// TIA Portal V17 program export: 1 tag tables, 1 data types, 1 data blocks, 3 code blocks (in call order from the OBs), 1 instance data blocks

VAR_GLOBAL   // PLC tag table "IO_CC_Cav_A"
   O_CC_Coupelle_Up_Cav_A AT %Q600.7 : Bool;
   I_CC_TyrePresent_Pos_2_Cav_A AT %I600.2 : Bool;
   I_CC_TyrePresent_Pos_3_Cav_A AT %I600.3 : Bool;
   I_CC_TyrePresent_Coupelle_Cav_A AT %I600.0 : Bool;
   I_CC_TyrePresent_Exit_Cav_A AT %I600.1 : Bool;
   I_CC_Coupelle_Low_Cav_A AT %I600.4 : Bool;
   I_CC_Coupelle_High_Cav_A AT %I600.5 : Bool;
   I_CC_Motor_Lototo_Cav_A AT %I600.6 : Bool;
   O_CC_Coupelle_Down_Cav_A AT %Q601.7 : Bool;
   I_CC_TyrePresent_Pos_1_Cav_A AT %I601.0 : Bool;
END_VAR

TYPE "CAB"
// stored: IsFailsafeCompliant false
   STRUCT
      CAB : String[20];
   END_STRUCT;
END_TYPE

DATA_BLOCK "GlobalData"   // DB1
{ S7_Optimized_Access := 'TRUE' }
VERSION : 0.1
// stored: AutoNumber true, IsIECCheckEnabled false
   VAR
      Ready : Bool;
      Count : Int;
      Config : Struct
         MaxSpeed : Real;
         Enabled : Bool;
      END_STRUCT;
   END_VAR
BEGIN
END_DATA_BLOCK

ORGANIZATION_BLOCK "Main"   // OB1, LAD, ProgramCycle
TITLE = "Main Program Sweep (Cycle)"
{ S7_Optimized_Access := 'TRUE' }
VERSION : 0.1
// stored: AutoNumber true, IsIECCheckEnabled false, SetENOAutomatically false
   VAR_INPUT
      Initial_Call : Bool;   // Initial call of this OB
      Remanence : Bool;   // =True, if remanent data are available
   END_VAR
BEGIN

REGION Network 1
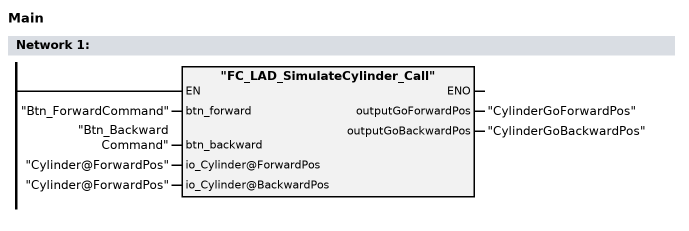
   RUNG wire#powerrail
      "FC_LAD_SimulateCylinder_Call"(btn_forward := "Btn_ForwardCommand", btn_backward := "Btn_BackwardCommand", "io_Cylinder@ForwardPos" := "Cylinder@ForwardPos", "io_Cylinder@BackwardPos" := "Cylinder@ForwardPos", outputGoForwardPos => "CylinderGoForwardPos", outputGoBackwardPos => "CylinderGoBackwardPos")
   END_RUNG
   // the same network as SCL:
   "FC_LAD_SimulateCylinder_Call"(btn_forward := "Btn_ForwardCommand",
                           btn_backward := "Btn_BackwardCommand",
                           "io_Cylinder@ForwardPos" := "Cylinder@ForwardPos",
                           "io_Cylinder@BackwardPos" := "Cylinder@ForwardPos",
                           outputGoForwardPos => "CylinderGoForwardPos",
                           outputGoBackwardPos => "CylinderGoBackwardPos");
END_REGION
END_ORGANIZATION_BLOCK

FUNCTION "FC_LAD_SimulateCylinder_Call" : Void   // FC1, LAD
{ S7_Optimized_Access := 'TRUE' }
VERSION : 0.1
// stored: AutoNumber true, IsIECCheckEnabled false, SetENOAutomatically false, UDAEnableTagReadback false
   VAR_INPUT
      btn_forward : Bool;
      btn_backward : Bool;
   END_VAR
   VAR_OUTPUT
      outputGoForwardPos : Bool;
      outputGoBackwardPos : Bool;
   END_VAR
   VAR_IN_OUT
      "io_Cylinder@ForwardPos" : Bool;
      "io_Cylinder@BackwardPos" : Bool;
   END_VAR
BEGIN

REGION Network 1
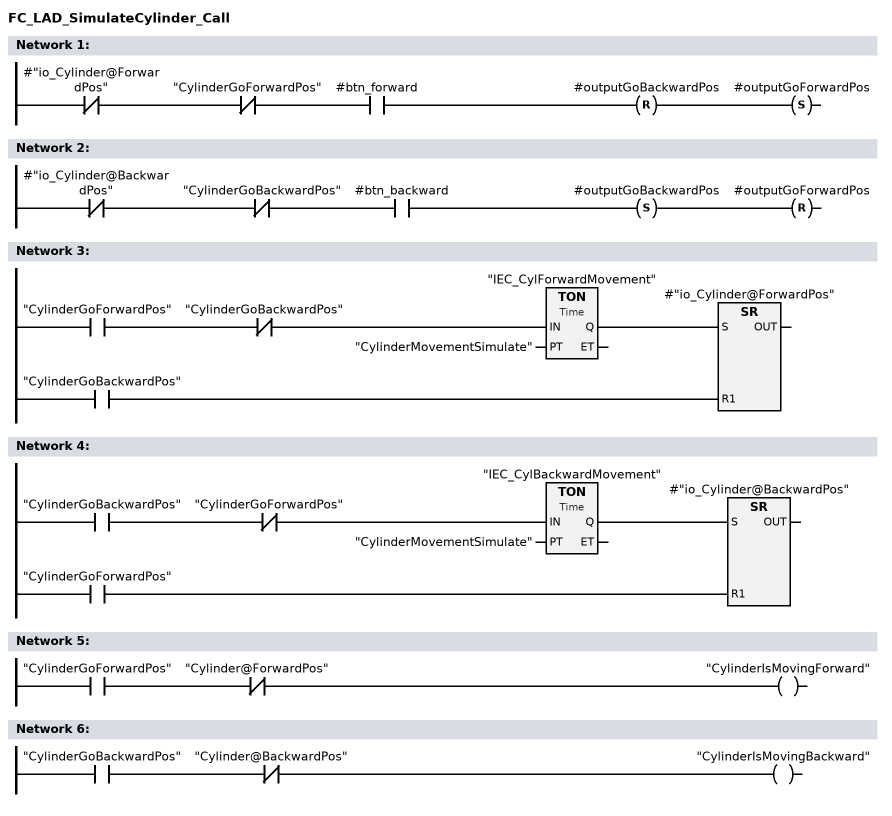
   RUNG wire#powerrail
      I_Contact( #"io_Cylinder@ForwardPos" )
      I_Contact( "CylinderGoForwardPos" )
      Contact( #btn_forward )
      R_Coil( #outputGoBackwardPos )
      S_Coil( #outputGoForwardPos )
   END_RUNG
   // the same network as SCL:
   IF NOT #"io_Cylinder@ForwardPos" AND NOT "CylinderGoForwardPos" AND #btn_forward THEN
       #outputGoBackwardPos := FALSE;
       #outputGoForwardPos := TRUE;
   END_IF;
END_REGION

REGION Network 2
   RUNG wire#powerrail
      I_Contact( #"io_Cylinder@BackwardPos" )
      I_Contact( "CylinderGoBackwardPos" )
      Contact( #btn_backward )
      S_Coil( #outputGoBackwardPos )
      R_Coil( #outputGoForwardPos )
   END_RUNG
   // the same network as SCL:
   IF NOT #"io_Cylinder@BackwardPos" AND NOT "CylinderGoBackwardPos" AND #btn_backward THEN
       #outputGoBackwardPos := TRUE;
       #outputGoForwardPos := FALSE;
   END_IF;
END_REGION

REGION Network 3
   RUNG wire#powerrail
      Contact( "CylinderGoForwardPos" )
      I_Contact( "CylinderGoBackwardPos" )
      { S7_Templates := "time_type := Time" } "IEC_CylForwardMovement".TON(pt := "CylinderMovementSimulate", et =>)
      S_SR(operand := #"io_Cylinder@ForwardPos", r1 := wire#w1)
   END_RUNG
   RUNG wire#powerrail
      Contact( "CylinderGoBackwardPos" )
   END_RUNG wire#w1
   // the same network as SCL:
   "IEC_CylForwardMovement".TON(IN := "CylinderGoForwardPos" AND NOT "CylinderGoBackwardPos",
                           PT := "CylinderMovementSimulate");
   IF "IEC_CylForwardMovement".Q THEN
       #"io_Cylinder@ForwardPos" := TRUE;   // SR flip-flop
   END_IF;
   IF "CylinderGoBackwardPos" THEN #"io_Cylinder@ForwardPos" := FALSE; END_IF;
END_REGION

REGION Network 4
   RUNG wire#powerrail
      Contact( "CylinderGoBackwardPos" )
      I_Contact( "CylinderGoForwardPos" )
      { S7_Templates := "time_type := Time" } "IEC_CylBackwardMovement".TON(pt := "CylinderMovementSimulate", et =>)
      S_SR(operand := #"io_Cylinder@BackwardPos", r1 := wire#w1)
   END_RUNG
   RUNG wire#powerrail
      Contact( "CylinderGoForwardPos" )
   END_RUNG wire#w1
   // the same network as SCL:
   "IEC_CylBackwardMovement".TON(IN := "CylinderGoBackwardPos" AND NOT "CylinderGoForwardPos",
                           PT := "CylinderMovementSimulate");
   IF "IEC_CylBackwardMovement".Q THEN
       #"io_Cylinder@BackwardPos" := TRUE;   // SR flip-flop
   END_IF;
   IF "CylinderGoForwardPos" THEN #"io_Cylinder@BackwardPos" := FALSE; END_IF;
END_REGION

REGION Network 5
   RUNG wire#powerrail
      Contact( "CylinderGoForwardPos" )
      I_Contact( "Cylinder@ForwardPos" )
      Coil( "CylinderIsMovingForward" )
   END_RUNG
   // the same network as SCL:
   "CylinderIsMovingForward" := "CylinderGoForwardPos" AND NOT "Cylinder@ForwardPos";
END_REGION

REGION Network 6
   RUNG wire#powerrail
      Contact( "CylinderGoBackwardPos" )
      I_Contact( "Cylinder@BackwardPos" )
      Coil( "CylinderIsMovingBackward" )
   END_RUNG
   // the same network as SCL:
   "CylinderIsMovingBackward" := "CylinderGoBackwardPos" AND NOT "Cylinder@BackwardPos";
END_REGION
END_FUNCTION

FUNCTION "SclAssign" : Void   // FC10, SCL
VERSION : 0.1
// stored: AutoNumber true, IsIECCheckEnabled false
BEGIN

REGION Network 1: Write counters
   "GlobalData".Count := "GlobalData".Ready;
   "GlobalData".Config.MaxSpeed := "GlobalData".Count;
END_REGION

REGION Network 2: Gate ready flag
   IF "GlobalData".Config.Enabled THEN
   "GlobalData".Ready := FALSE;
   END_IF;
END_REGION
END_FUNCTION

DATA_BLOCK "MotorFbInstance"   // DB2
{ S7_Optimized_Access := 'TRUE' }
VERSION : 0.1
// stored: AutoNumber true, InstanceOfName MotorFb, IsIECCheckEnabled false
"MotorFb"
   // VAR
   //    Running : Bool;
   //    Setpoint : Real;
   // END_VAR
BEGIN
END_DATA_BLOCK
